// TIA Portal V17 export
// export: Created 2025-03-05T08:01:42.9765217Z, ExportSetting WithDefaults, DisplayName Totally Integrated Automation Portal, DisplayVersion V17 Update 8, DisplayName TIA Portal Openness, DisplayVersion V17 Update 8, DisplayName TIA Portal Version Control Interface, DisplayVersion V17, DisplayName SINAMICS Startdrive Advanced, DisplayVersion V17 SP2, DisplayName SINAMICS Startdrive G110M, G120, G120C, G120D, G120P, G115D, DisplayVersion V17 SP2, DisplayName SINAMICS Startdrive G130, G150, S120, S150, SINAMICS MV, S210, DisplayVersion V17 SP2, DisplayName STEP 7 Professional, DisplayVersion V17 Update 8, DisplayName SINUMERIK ONE STEP 7 Toolbox, DisplayVersion V17 Update 12, DisplayName SINUMERIK 840D sl STEP 7 Toolbox, DisplayVersion V17 Update 12, DisplayName STEP 7 Safety, DisplayVersion V17 Update 6, DisplayName WinCC Advanced, DisplayVersion V17 Update 8
DATA_BLOCK "DB7217_TRADES_CALL"   // DB7217
{ S7_Optimized_Access := 'FALSE'; DB_Accessible_From_OPC_UA := 'FALSE' }
AUTHOR : ETXETAR
VERSION : 1.0
// stored: AutoNumber false, DBAccessibleFromOPCUA false, DBAccessibleFromWebserver true, IsOnlyStoredInLoadMemory false, IsWriteProtectedInAS false
   VAR RETAIN
      GENERAL_CONDITIONS : Bool;   // GENERAL CONDITIONS
      I_1 : Bool;   // I 1
      I_2 : Bool;   // I 2
      I_3 : Bool;   // I 3
      I_4 : Bool;   // I 4
      I_5 : Bool;   // I 5
      I_6 : Bool;   // I 6
      I_7 : Bool;   // I 7
      CALL_1_REQ : Bool;   // CALL 1 REQUEST / CALL 1 REQ
      CANCEL_1_REQ : Bool;   // CANCEL 1 REQUEST / CANCEL 1 REQ
      CALL_2_REQ : Bool;   // CALL 2 REQUEST / CALL 2 REQ
      CANCEL_2_REQ : Bool;   // CANCEL 2 REQUEST / CANCEL 2 REQ
      CALL_3_REQ : Bool;   // CALL 3 REQUEST / CALL 3 REQ
      CANCEL_3_REQ : Bool;   // CANCEL 3 REQUEST / CANCEL 3 REQ
      CALL_4_REQ : Bool;   // CALL 4 REQUEST / CALL 4 REQ
      CANCEL_4_REQ : Bool;   // CANCEL 4 REQUEST / CANCEL 4 REQ
      CALL_5_REQ : Bool;   // CALL 5 REQUEST / CALL 5 REQ
      CANCEL_5_REQ : Bool;   // CANCEL 5 REQUEST / CANCEL 5 REQ
      CALL_6_REQ : Bool;   // CALL 6 REQUEST / CALL 6 REQ
      CANCEL_6_REQ : Bool;   // CANCEL 6 REQUEST / CANCEL 6 REQ
      CALL_7_REQ : Bool;   // CALL 7 REQUEST / CALL 7 REQ
      CANCEL_7_REQ : Bool;   // CANCEL 7 REQUEST / CANCEL 7 REQ
      CALL_8_REQ : Bool;   // CALL 8 REQUEST / CALL 8 REQ
      CANCEL_8_REQ : Bool;   // CANCEL 8 REQUEST / CANCEL 8 REQ
      CALL_1 : Bool;   // CALL #1 / CALL 1
      CALL_2 : Bool;   // CALL #2 / CALL 2
      CALL_3 : Bool;   // CALL #3 / CALL 3
      CALL_4 : Bool;   // CALL #4 / CALL 4
      CALL_5 : Bool;   // CALL #5 / CALL 5
      CALL_6 : Bool;   // CALL #6 / CALL 6
      CALL_7 : Bool;   // CALL #7 / CALL 7
      CALL_8 : Bool;   // CALL 8
      CALL_1_AUX : Bool;   // CALL 1 AUX
      CALL_2_AUX : Bool;   // CALL 2 AUX
      CALL_3_AUX : Bool;   // CALL 3 AUX
      CALL_4_AUX : Bool;   // CALL 4 AUX
      CALL_5_AUX : Bool;   // CALL 5 AUX
      CALL_6_AUX : Bool;   // CALL 6 AUX
      CALL_7_AUX : Bool;   // CALL 7 AUX
      CALL_8_AUX : Bool;   // CALL 8 AUX
      CALL_1_ACK_AUX : Bool;   // CALL 1 ACK AUX
      CALL_2_ACK_AUX : Bool;   // CALL 2 ACK AUX
      CALL_3_ACK_AUX : Bool;   // CALL 3 ACK AUX
      CALL_4_ACK_AUX : Bool;   // CALL 4 ACK AUX
      CALL_5_ACK_AUX : Bool;   // CALL 5 ACK AUX
      CALL_6_ACK_AUX : Bool;   // CALL 6 ACK AUX
      CALL_7_ACK_AUX : Bool;   // CALL 7 ACK AUX
      CALL_8_ACK_AUX : Bool;   // CALL 8 ACK AUX
      CALL_1_ACKNOWLEDGE : Bool;   // CALL 1 ACKNOWLEDGE
      CALL_2_ACKNOWLEDGE : Bool;   // CALL 2 ACKNOWLEDGE
      CALL_3_ACKNOWLEDGE : Bool;   // CALL 3 ACKNOWLEDGE
      CALL_4_ACKNOWLEDGE : Bool;   // CALL 4 ACKNOWLEDGE
      CALL_5_ACKNOWLEDGE : Bool;   // CALL 5 ACKNOWLEDGE
      CALL_6_ACKNOWLEDGE : Bool;   // CALL 6 ACKNOWLEDGE
      CALL_7_ACKNOWLEDGE : Bool;   // CALL 7 ACKNOWLEDGE
      CALL_8_ACKNOWLEDGE : Bool;   // CALL 8 ACKNOWLEDGE
      IS : Bool;   // IMMEDIATE STOP ALARMS / IS
      IS_SEOC : Bool;   // IMMEDIATE STOP & STOP AT END OF CYCLE ALARMS / IS SEOC
      RHP : Bool;   // RETURN TO HOME POSITION ALARMS / RHP
      RHP_SEOC : Bool;   // RETURN TO HOME POSITION & STOP AT END OF CYCLE ALARMS / RHP SEOC
      SEOC : Bool;   // STOP AT END OF CYCLE ALARMS / SEOC
      IS_WARNING : Bool;   // IMMEDIATE STOP WARNING / IS WARNING
      RHP_WARNING : Bool;   // RETURN TO HOME POSITION WARNING / RHP WARNING
      SEOC_WARNING : Bool;   // STOP AT END OF CYCLE WARNING / SEOC WARNING
      WARNING : Bool;   // WARNING
      HELP : Bool;   // HELP
      SP8_2 : Bool;   // SP8 2
      SP8_3 : Bool;   // SP8 3
      SP8_4 : Bool;   // SP8 4
      SP8_5 : Bool;   // SP8 5
      SP8_6 : Bool;   // SP8 6
      SP8_7 : Bool;   // SP8 7
      PULSE_1 : Bool;   // PULSE 1
      PULSE_2 : Bool;   // PULSE 2
      PULSE_3 : Bool;   // PULSE 3
      PULSE_4 : Bool;   // PULSE 4
      PULSE_5 : Bool;   // PULSE 5
      PULSE_6 : Bool;   // PULSE 6
      PULSE_7 : Bool;   // PULSE 7
      PULSE_8 : Bool;   // PULSE 8
      PULSE_9 : Bool;
      PULSE_10 : Bool;
      PULSE_11 : Bool;
      PULSE_12 : Bool;
      PULSE_13 : Bool;
      PULSE_14 : Bool;
      PULSE_15 : Bool;
      PULSE_16 : Bool;
      CALL_1_ACK : Bool;   // CALL 1 ACK
      CALL_2_ACK : Bool;   // CALL 2 ACK
      CALL_3_ACK : Bool;   // CALL 3 ACK
      CALL_4_ACK : Bool;   // CALL 4 ACK
      CALL_5_ACK : Bool;   // CALL 5 ACK
      CALL_6_ACK : Bool;   // CALL 6 ACK
      CALL_7_ACK : Bool;   // CALL 7 ACK
      CALL_8_ACK : Bool;   // CALL 8 ACK
      COUNT_CALL_NUM_1 : Int;   // COUNT CALL NUM 1
      COUNT_CALL_NUM_2 : Int;   // COUNT CALL NUM 2
      COUNT_CALL_NUM_3 : Int;   // COUNT CALL NUM 3
      COUNT_CALL_NUM_4 : Int;   // COUNT CALL NUM 4
      COUNT_CALL_NUM_5 : Int;   // COUNT CALL NUM 5
      COUNT_CALL_NUM_6 : Int;   // COUNT CALL NUM 6
      COUNT_CALL_NUM_7 : Int;   // COUNT CALL NUM 7
      COUNT_CALL_NUM_8 : Int;   // COUNT CALL NUM 8
   END_VAR
BEGIN
END_DATA_BLOCK
